FUNCTION RND (* this function rounds a real to n significant digits (not digits behind the comma). *)
  (* Standard: 61499-1 *)
  (* Version 1.0, 2026-09-17, Franz Höpfinger, Portiert aus OSCAT_basic RND.TcPOU - EXPT(10.0, ...) mit Begrenzung N (1..8), Exponenten-LIMIT (-37..8) und Bereichspruefung (ABS(X * M) >= 2.147e9) schuetzt vor DINT-Ueberlauf und Division durch 0. *)
  PACKAGE OSCAT::Basic::POUs::Mathematical;
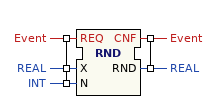
  EVENT_INPUT
    REQ WITH X, N;
  END_EVENT
  EVENT_OUTPUT
    CNF WITH RND;
  END_EVENT
  VAR_INPUT
    X : REAL;
    N : INT;
  END_VAR
  VAR_OUTPUT
    RND : REAL;
  END_VAR
  BODY IN ST:
PACKAGE OSCAT::Basic::POUs::Mathematical;

(* this function rounds a real to n significant digits (not digits behind the comma). *)
FUNCTION RND : REAL
VAR_INPUT
	X : REAL;
	N : INT;
END_VAR
VAR
	M : REAL;
END_VAR

(*
 * version 1.1	4. apr. 2008 programmer 	hugo tested by	tobias
 * *
 * this function rounds x to n significant digits.
 * unlike round(), n is not the number of digits behind the comma but the total number of
 * significant digits.
 * Portiert 2026-09-17: Begrenzung N (1..8), Exponenten-LIMIT (-37..8) und Bereichspruefung schuetzen vor DINT-Ueberlauf.
 *)
IF X = 0.0 THEN
	RND := 0.0;
ELSE
	M := EXPT(10.0, LIMIT(-37.0, INT_TO_REAL(LIMIT(1, N, 8)) - CEIL(LOG(ABS(X))), 8.0));
	IF ABS(X * M) >= 2147483647.0 THEN
		RND := X;
	ELSE
		RND := DINT_TO_REAL(REAL_TO_DINT(X * M)) / M;
	END_IF;
END_IF;

END_FUNCTION

(* revision history hm	1. sep 2006	rev 1.0 original version
 * *
 * hm	4. apr. 2008	rev 1.1 added type conversion to avoid warning under codesys 3.0 *)
  END_BODY
END_FUNCTION
